{attribute addProperty BoxType "EL5151-0021-0018"}
{attribute addProperty Id "ENC_StatusAT %I*ENC_Status_053BC81D80100ENC_Filtered_latchAT %I*ENC_Filtered_latch_7F6716946480ENC_ControlAT %Q*ENC_Control_E047A95D112140WcStateAT %I*WcState_F855686C1620InfoDataAT %I*InfoData_BC63D37F80100"}
{attribute addProperty CRC "1302125415"}
{attribute addProperty SizeInBites "352"}
{attribute addProperty SizeInBytes "44"}
TYPE EL5151_B58C1E49 :
STRUCT
	{attribute addProperty Name "ENC_Status"}
	ENC_Status : ENC_Status_053BC81D;
	{attribute addProperty Name "ENC_Filtered_latch"}
	ENC_Filtered_latch : ENC_Filtered_latch_7F671694;
	{attribute addProperty Name "ENC_Control"}
	ENC_Control : ENC_Control_E047A95D;
	{attribute addProperty Name "WcState"}
	WcState : WcState_F855686C;
	{attribute addProperty Name "InfoData"}
	InfoData : InfoData_BC63D37F;
END_STRUCT
END_TYPE

(* stored: Version 1.2.0.0, ProductVersion 3.1.4024.9
   DUT EL5151_B58C1E49: Id {5a63a5c4-7285-461b-83e9-461d578a80d3} *)
